(* Logix 5000 project; controller CambioGiroMotor vendor 1 type 14 code 156 rev 30.11; software revision 30.00 *)

TASK MainTask (continuous, watchdog 500 ms) : MainProgram

MODULES
   Local : vendor 1 type 14 code 156 (Compact 0, rev 30.11)
      DIG_IN : 1769-IQ16 (Compact 4, rev 1.1, Input RPI 20 ms)
      ANALOG_OUT : vendor 1 type 10 code 48 (Compact 3, rev 1.1, Output RPI 80 ms)
      DIG_OUT : vendor 1 type 7 code 86 (Compact 5, rev 2.1, Output RPI 20 ms)
      ANALOG_IN : vendor 1 type 10 code 44 (Compact 2, rev 2.1, Output RPI 80 ms)
      DEVICENET : vendor 1 type 12 code 105 (Compact 1, rev 1.1, Output RPI 20 ms)
END_MODULES

VAR_GLOBAL   (* controller tags *)
   GD_OUT_0 : BOOL;
   GD_OUT_1 : BOOL;
   Prueba : BOOL;
END_VAR

PROGRAM MainProgram   (* main routine MainRoutine *)
VAR
   km1 : ALIAS FOR Local:5:O.Data.0;
   km2 : ALIAS FOR Local:4:I.Data.1;
   star_der : ALIAS FOR Local:4:I.Data.3;
   start : ALIAS FOR Local:4:I.Data.1;
   start_izq : ALIAS FOR Local:4:I.Data.2;
   stop : ALIAS FOR Local:4:I.Data.0;
END_VAR

ROUTINE MainRoutine   (* ladder *)
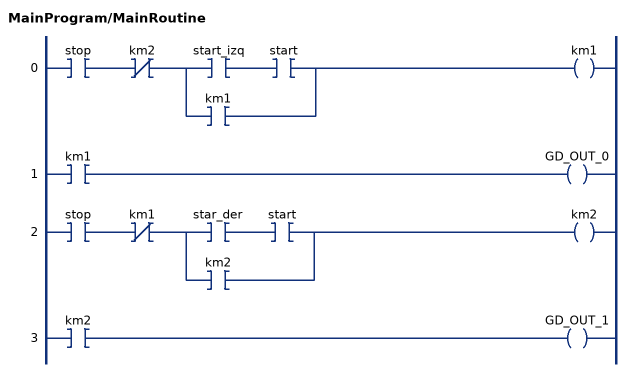
   0: XIC(stop)XIO(km2)[XIC(start_izq) XIC(start) ,XIC(km1) ]OTE(km1);
   1: XIC(km1)OTE(GD_OUT_0);
   2: XIC(stop)XIO(km1)[XIC(star_der) XIC(start) ,XIC(km2) ]OTE(km2);
   3: XIC(km2)OTE(GD_OUT_1);
END_ROUTINE
END_PROGRAM
